FUNCTION Updete_Motor_Parameters
VAR_INPUT
	bUpdateValue : BOOL;
	fNewValue : REAL;
	stMotorParameters : ST_Motor;
END_VAR
VAR
END_VAR

IF bUpdateValue = 1 THEN
	stMotorParameters.fSpeedMax := fNewValue;
ELSE
	stMotorParameters.fSpeedMax := stMotorParameters.fSpeedMax;
END_IF

END_FUNCTION

(* stored: Version 1.1.0.1, ProductVersion 3.1.4024.12
   POU Updete_Motor_Parameters: Id {5fa040b2-2604-4c24-b503-c574900a23c8}, SpecialFunc None *)
